KUKA KRL data list: dockon_3.dat

&ACCESS RV1
&REL 138
&COMMENT PICKUP GUN 3
DEFDAT  DOCKON_3
;FOLD EXTERNAL DECLARATIONS;%{PE}%MKUKATPBASIS,%CEXT,%VCOMMON,%P
;FOLD GRIPPERTECH EXT
EXT  H50 (INT  :IN,INT  :IN,INT  :IN,GRP_TYP  :IN )
;ENDFOLD (GRIPPERTECH EXT)
;FOLD SPOTTECH EXT
EXT  USERSPOT (S_COMMAND  :IN,SPOT_TYPE  :IN )
;ENDFOLD (SPOTTECH EXT)
;FOLD BASISTECH EXT;%{PE}%MKUKATPBASIS,%CEXT,%VEXT,%P
EXT  BAS (BAS_COMMAND  :IN,REAL  :IN )
DECL INT SUCCESS
;ENDFOLD (BASISTECH EXT)
;FOLD USER EXT;%{E}%MKUKATPUSER,%CEXT,%VEXT,%P
;Make here your modifications
;ENDFOLD (USER EXT)
;ENDFOLD (EXTERNAL DECLERATIONS)
DECL GRP_TYP GCONT={G_APO #YES,TIME 0.0,CTRL #OFF,DLY 0,DST 0}
DECL GRP_TYP GGDAT={G_APO #NO,TIME 0.0,CTRL #OFF,DLY 0,DST 1}
;*      FDAT Declarations     *

;******************************
;*     E6POS Declarations     *
;******************************

DECL E6POS XP10={X -1127.36902,Y 2445.76807,Z 816.869385,A -45.7330017,B 0.4947837,C 179.7724,S 2,T 11,E1 -1181.96399,E2 0.0,E3 0.0,E4 0.0,E5 0.0,E6 0.0}
DECL E6POS XP20={X -1446.12402,Y 3116.53906,Z 717.922974,A 58.8610001,B -0.318507999,C -179.604202,S 2,T 3,E1 -1703.68103,E2 0.0,E3 0.0,E4 0.0,E5 0.0,E6 0.0}
DECL E6POS XP30={X -1433.29297,Y 3103.76904,Z 492.324188,A 58.8653107,B -0.296647787,C -179.599304,S 2,T 3,E1 -1703.68103,E2 0.0,E3 0.0,E4 0.0,E5 0.0,E6 0.0}
DECL E6POS XP40={X -1433.297,Y 3103.77197,Z 406.572693,A 58.865181,B -0.296665102,C -179.598999,S 2,T 3,E1 -1703.68103,E2 0.0,E3 0.0,E4 0.0,E5 0.0,E6 0.0}
DECL E6POS XP50={X -1220.43506,Y 3106.93091,Z -694.426208,A -13.5916004,B 72.6322479,C -12.8654499,S 2,T 3,E1 -1703.68298,E2 0.0,E3 0.0,E4 0.0,E5 0.0,E6 0.0}
DECL E6POS XP60={X -1178.72095,Y 3107.79907,Z -662.205017,A -13.5877895,B 72.6321716,C -12.8613501,S 2,T 3,E1 -1703.68298,E2 0.0,E3 0.0,E4 0.0,E5 0.0,E6 0.0}
DECL E6POS XP70={X -1104.13306,Y 3107.021,Z -353.061005,A -13.5874701,B 72.6343613,C -12.8619604,S 2,T 3,E1 -1703.68506,E2 0.0,E3 0.0,E4 0.0,E5 0.0,E6 0.0}
DECL E6POS XP80={X -889.438477,Y 2792.34302,Z 1049.42505,A -106.691704,B 85.8009872,C -106.606796,S 2,T 11,E1 -1703.68701,E2 0.0,E3 0.0,E4 0.0,E5 0.0,E6 0.0}

;******************************
;*     FDAT Declarations      *
;******************************

DECL FDAT FP10={TOOL_NO 10,BASE_NO 0,IPO_FRAME #BASE}
DECL FDAT FP20={TOOL_NO 10,BASE_NO 0,IPO_FRAME #BASE}
DECL FDAT FP30={TOOL_NO 10,BASE_NO 0,IPO_FRAME #BASE}
DECL FDAT FP40={TOOL_NO 10,BASE_NO 0,IPO_FRAME #BASE}
DECL FDAT FP50={TOOL_NO 3,BASE_NO 0,IPO_FRAME #BASE}
DECL FDAT FP60={TOOL_NO 3,BASE_NO 0,IPO_FRAME #BASE}
DECL FDAT FP70={TOOL_NO 3,BASE_NO 0,IPO_FRAME #BASE}
DECL FDAT FP80={TOOL_NO 3,BASE_NO 0,IPO_FRAME #BASE}

;******************************
;*  PDAT & LDAT Declarations  *
;******************************

DECL PDAT PH={VEL 100.0,ACC 100.0,APO_DIST 100.0}
DECL LDAT LH={VEL 2.0,ACC 100.0,APO_DIST 100.0,APO_FAC 50.0,ORI_TYP #VAR}

DECL E6POS XP1={X -1220.39795,Y 3105.43091,Z -744.515076,A -13.7468996,B 72.6471634,C -12.8395901,S 2,T 3,E1 -1701.58704,E2 0.0,E3 0.0,E4 0.0,E5 0.0,E6 0.0}
DECL FDAT FP1={TOOL_NO 3,BASE_NO 0,IPO_FRAME #BASE,POINT2[] " "}
DECL PDAT PPDAT1={VEL 100.0,ACC 100.0,APO_DIST 100.0}
ENDDAT
